PROGRAM EM01_Master
VAR
	ref_Master1: REFERENCE TO UDT_AXISADMIN;	
	ref_Follower4: REFERENCE TO UDT_AXISADMIN;
	ref_Follower5: REFERENCE TO UDT_AXISADMIN;	
	Ref_MachineStateModel: REFERENCE TO PackMlv3_StateModel;
	ref_Work_Recipe: REFERENCE TO UDT_Hmi_Output; //当前生产的配方

    Ref_Unit: REFERENCE TO UDT_UnitAdmin;
	ref_lrLatchMasterPos: REFERENCE TO LREAL;
	ref_BinList: REFERENCE TO UDT_BINlist;	
	ref_diBeltObjCnt: REFERENCE TO DINT;
	EM_No: INT:=1;

	tonAbortingWatchDog: TON;   
	MasterSeq: SequenceTransfer;
	
END_VAR

VAR CONSTANT

END_VAR

// 主轴走200MM产出一个产品
Ref_MachineStateModel REF= UN01_MachineStateModel;
Ref_Unit REF=Unit01;
ref_Work_Recipe REF= HMI_Output;
ref_Follower4  REF= arRealAxisAdmin[44];
ref_Follower5  REF= arRealAxisAdmin[45];
ref_Master1 REF= arVirtualAxisAdmin[1];

ref_BinList REF=Glb_BinList;
ref_diBeltObjCnt REF=glb_diBeltObjCnt;
CM01_Master();
MainRoution();
SR99_FaultHandle();

ref_master1.i.PosRangeTable[1][1]:=190;
ref_master1.i.PosRangeTable[1][2]:=200;

ACTION CM01_Master:
CASE MasterSeq.Now OF		 
	0: 
	   IF Ref_MachineStateModel.Sts_Resetting THEN
		  MasterSeq(ExeCute:= TRUE, Next:= Seq_Resetting );
	   END_IF	   
	   IF Ref_MachineStateModel.Sts_Stopping  THEN
          MasterSeq(ExeCute:= TRUE, Next:= Seq_StoppingDone );  
	   END_IF	

	Seq_Resetting:
		IF NOT ref_Master1.o.PowerOn  THEN;
		   ref_Master1.i.Enable:=TRUE;
	    ELSE
		   MasterSeq(ExeCute:= TRUE, Next:= 20 );
		END_IF
	    IF Ref_MachineStateModel.Sts_Stopping  THEN
		   MasterSeq(ExeCute:= TRUE, Next:= Seq_Stopping);  
	    END_IF	
	20:	
	       ref_master1.i.PosRangeTable[1][1]:=0;
		   ref_master1.i.PosRangeTable[1][2]:=10;
		   ref_master1.i.JogAcc:=100;
		   ref_Master1.i.JogDec:=5000;
		   IF NOT glb_AllAxisHomed_UN01 THEN
			  MasterSeq(ExeCute:= TRUE, Next:= 21 );
			  ELSE
			  MasterSeq(ExeCute:= TRUE, Next:= Seq_ResettingDone );
		   END_IF
	21:    
		   ref_Master1.i.HomeMode:=2;
		   ref_Master1.i.Home:=TRUE;
		   IF ref_Master1.o.HomeDone THEN
			   ref_Master1.i.Home:=FALSE;
			   MasterSeq(ExeCute:= TRUE, Next:= 30 );
		   ELSE IF Ref_MachineStateModel.Sts_Stopping  THEN
		           MasterSeq(ExeCute:= TRUE, Next:= Seq_Stopping);  
	            END_IF	 
		   END_IF
    30:   

		  glb_diBeltObjCnt:=0;
          MasterSeq(ExeCute:= TRUE, Next:= Seq_ResettingDone ); 
		  
	Seq_ResettingDone: 
         IF NOT Ref_MachineStateModel.Sts_Resetting THEN
			MasterSeq(ExeCute:= TRUE, Next:= 0 );
		 END_IF	  
 	  
	Seq_Stopping:	
	     MasterSeq(ExeCute:= TRUE, Next:= Seq_StoppingDone); 
	Seq_StoppingDone: 
	     IF NOT Ref_MachineStateModel.Sts_Stopping THEN
			MasterSeq(ExeCute:= TRUE, Next:= 0 );
		 END_IF	   
		 
END_CASE
MasterSeq(ExeCute:= FALSE, Next:= , Last=> , Now=> );
END_ACTION

ACTION MainRoution:
EM_No:=1;
IF Ref_Unit.EM_Selected[EM_No] THEN
	IF Ref_MachineStateModel.Sts_Holding THEN
		Ref_Unit.EM_Holding_Done[EM_No]:=TRUE;
		ELSE
		Ref_Unit.EM_Holding_Done[EM_No]:=FALSE;
	END_IF
	IF Ref_MachineStateModel.Sts_UnHolding THEN
		Ref_Unit.EM_UnHolding_Done[EM_No]:=TRUE;
		ELSE
		Ref_Unit.EM_UnHolding_Done[EM_No]:=FALSE;
	END_IF
	
	IF Ref_MachineStateModel.Sts_Suspending THEN
		Ref_Unit.EM_Suspending_Done[EM_No]:=TRUE;
		ELSE
		Ref_Unit.EM_Suspending_Done[EM_No]:=FALSE;
	END_IF
	
	IF Ref_MachineStateModel.Sts_UnSuspending THEN
		Ref_Unit.EM_UnSuspending_Done[EM_No]:=TRUE;
		ELSE
		Ref_Unit.EM_UnSuspending_Done[EM_No]:=FALSE;
	END_IF
		
	IF Ref_MachineStateModel.Sts_Resetting AND MasterSeq.Now=Seq_ResettingDone  THEN
	   Ref_Unit.EM_Resetting_Done[EM_No]:=TRUE; 
       ELSE   
	   Ref_Unit.EM_Resetting_Done[EM_No]:=FALSE;
	END_IF
	
	IF Ref_MachineStateModel.Sts_Clearing THEN
	      Ref_Unit.EM_Clearing_Done[EM_No]:=TRUE;
		  ELSE
		  Ref_Unit.EM_Clearing_Done[EM_No]:=FALSE;
	END_IF
	
	IF Ref_MachineStateModel.Sts_Aborting THEN
	   MasterSeq(ExeCute:= TRUE, Next:= 0 );
       IF tonAbortingWatchDog.Q THEN
		  ref_Master1.i.Disable:=TRUE;
		  Ref_Unit.EM_Aborting_Done[EM_No]:=TRUE;
	   END_IF
	   ELSE
		  Ref_Unit.EM_Aborting_Done[EM_No]:=FALSE;
	END_IF
	tonAbortingWatchDog(IN:= Ref_MachineStateModel.Sts_Aborting, PT:=T#3S , Q=> , ET=> );
	
	IF Ref_MachineStateModel.Sts_Starting THEN
	   Ref_Unit.EM_Starting_Done[EM_No]:=TRUE;
	   ELSE
	   Ref_Unit.EM_Starting_Done[EM_No]:=FALSE;
	END_IF
	
	IF Ref_MachineStateModel.Sts_Stopping  AND MasterSeq.Now=Seq_StoppingDone THEN
	   Ref_Unit.EM_Stopping_Done[EM_No]:=TRUE;
	   ELSE	   
	   Ref_Unit.EM_Stopping_Done[EM_No]:=FALSE;
	END_IF

END_IF
END_ACTION

ACTION SR99_FaultHandle:
;
END_ACTION

END_PROGRAM

(* stored: Version 1.1.0.1, ProductVersion 3.1.4024.6
   POU EM01_Master: Id {40be8088-7005-4369-a85a-46875fa0e609}, SpecialFunc None
   Action CM01_Master: Id {1ae91068-5d2b-4bbf-91cf-d600db16ff00}
   Action MainRoution: Id {529d5d32-328c-4e72-afd3-7b6c49aea43a}
   Action SR99_FaultHandle: Id {e7b41dea-36cd-4243-8903-31908f899a44} *)
